# B&R Automation Studio project lab2
Automation Studio 4.5.2.102

## Configuration SampleText

CPU 4PP065.0571-P74, AutomationRuntime D4.52, Build 4.1.2, Vc V4.25.0, Safety 1.6

### Task classes (Cpu.sw)
```
Cyclic#1 (cycle 2000 us, tolerance 0 us):
  ncsdcctrl <- ncsdcctrl.prg
Cyclic#4:
  DoorCtrl <- DoorCtrl.prg
  LED <- LED.prg
DataObjects: Acp10sys
NcDataObjects: acp10etxen <- acp10etxen.dob, gAxis01a <- gAxis01obj.gAxis01a.dob, gAxis01i <- gAxis01obj.gAxis01i.dob
Binaries: TCData, udbdef, iomap, arconfig, asfw, ashwac, sysconf, User, Role, ashwd, acp10cfg, Acp10map
Libraries: Acp10sdc, sys_lib, Runtime, asstring, Acp10man, Acp10par, NcGlobal, Acp10_MC, brsystem, AsBrStr, GateCtrl, astime, fileio, powerlnk, asieccon
```

### Hardware
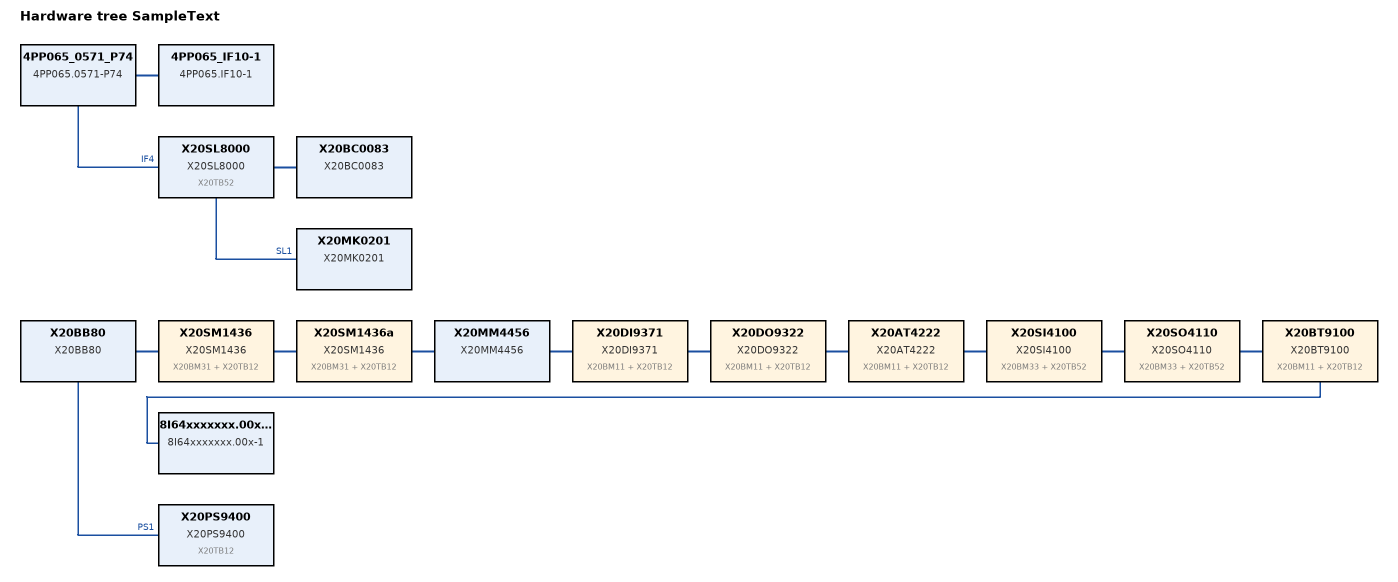
```
4PP065_0571_P74 : 4PP065.0571-P74 v1.1.2.0
  Connector IF4:
    EplInterfaceRedundant = 0
    EplEthInterfaceRedundant = 0
  Connector IF5:
    ActivateDevice = 1
    Mode = Manual
    InternetAddress = 10.0.1.1
    SubnetMask = 255.255.255.0
  ConfigurationID = labBR
  TimerDeviceType = EPLX2X
  TimerDevice = 4PP065_0571_P74.IF4
  TaskClassIdleTime = 2000
  Cyclic1Duration = 2000
  Cyclic1Tolerance = 0
  Cyclic1Output = 1
4PP065_IF10-1 : 4PP065.IF10-1 v1.0.3.0  [SS -> 4PP065_0571_P74.SS1]
8I64xxxxxxx.00x-1 : 8I64xxxxxxx.00x-1 v1.3.9.1  [X2X1 -> X20BT9100.X2X1 [Cable Type=X2XCable, Length=10, Version=1.0.0.2]]
  packedETAD = packed
  packedETI = packed
  packedCMDD = packed
  packedCMI = packed
  UNS = 220
  NCR = 10
  NSP = 890
  COS = 64
  RSC = 33000
X20AT4222 : X20AT4222 v1.2.3.0  [SS1 -> X20TB12e.SS; SL -> X20BM11c.SL1]
X20BB80 : X20BB80 v1.0.2.0
X20BC0083 : X20BC0083 v2.9.0.0  [PLK1 -> X20SL8000.PLK2 (NodeNumber=2) [Cable Type=PowerlinkCable, Length=10, Version=1.0.0.2]; SL -> X20BB80.SL1]
X20BM11 : X20BM11 v1.0.0.1  [X2X1 -> X20BM33a.X2X2]
X20BM11a : X20BM11 v1.0.0.1  [X2X1 -> X20MM4456.X2X2]
X20BM11b : X20BM11 v1.0.0.1  [X2X1 -> X20BM11a.X2X2]
X20BM11c : X20BM11 v1.0.0.1  [X2X1 -> X20BM11b.X2X2]
X20BM31 : X20BM31 v1.0.0.1  [X2X1 -> X20BB80.IF1]
X20BM31a : X20BM31 v1.0.0.1  [X2X1 -> X20BM31.X2X2]
X20BM33 : X20BM33 v1.0.0.4  [X2X1 -> X20BM11c.X2X2]
X20BM33a : X20BM33 v1.0.0.4  [X2X1 -> X20BM33.X2X2]
X20BT9100 : X20BT9100 v1.0.3.0  [SS1 -> X20TB12f.SS; SL -> X20BM11.SL1]
X20DI9371 : X20DI9371 v1.0.2.0  [SS1 -> X20TB12c.SS; SL -> X20BM11a.SL1]
X20DO9322 : X20DO9322 v1.0.3.0  [SS1 -> X20TB12d.SS; SL -> X20BM11b.SL1]
X20MK0201 : X20MK0201 v1.0.0.0  [SL -> X20SL8000.SL1]
X20MM4456 : X20MM4456 v1.1.5.0  [X2X1 -> X20BM31a.X2X2]
X20PS9400 : X20PS9400 v1.0.2.4  [SS1 -> X20TB12.SS; PS -> X20BB80.PS1]
X20SI4100 : X20SI4100 v1.10.1.1  [SS1 -> X20TB52.SS; SL -> X20BM33.SL1]
X20SL8000 : X20SL8000 v1.6.5.1  [PLK1 -> 4PP065_0571_P74.IF4 (NodeNumber=1) [Cable Type=PowerlinkCable, Length=10, Version=1.0.0.2]; PLK2 -> X20BC0083.PLK1 (NodeNumber=1) [Cable Type=PowerlinkCable, Length=10, Version=1.0.0.2]; SS1 -> X20TB52b.SS]
  SafeProject = SafeLOGIC-1
X20SM1436 : X20SM1436 v1.4.2.1  [SS1 -> X20TB12a.SS; SL -> X20BM31.SL1]
X20SM1436a : X20SM1436 v1.4.2.1  [SS1 -> X20TB12b.SS; SL -> X20BM31a.SL1]
X20SO4110 : X20SO4110 v1.10.1.1  [SS1 -> X20TB52a.SS; SL -> X20BM33a.SL1]
  SafeModuleID = 3
X20TB12 : X20TB12 v1.0.0.0
X20TB12a : X20TB12 v1.0.0.0
X20TB12b : X20TB12 v1.0.0.0
X20TB12c : X20TB12 v1.0.0.0
X20TB12d : X20TB12 v1.0.0.0
X20TB12e : X20TB12 v1.0.0.0
X20TB12f : X20TB12 v1.0.0.0
X20TB52 : X20TB52 v1.0.0.1
X20TB52a : X20TB52 v1.0.0.1
X20TB52b : X20TB52 v1.0.0.1
```

### IoMap.iom - 4PP065_0571_P74/IoMap.iom
```iecst
VAR_CONFIG
	Cyclic#1.gAxis01_DrvIf.iLifeCnt AT %IB."8I64xxxxxxx.00x-1".SDC_LifeCnt;
	Cyclic#1.gAxis01_DrvIf.iDrvOK AT %IX."8I64xxxxxxx.00x-1".ETAD_Input_Bool_02;
	Cyclic#1.gAxis01_DrvIf.oSetTime AT %QW."8I64xxxxxxx.00x-1".SDC_SetTime;
	Cyclic#1.::DoorCtrl:driveSM.speed AT %QW."8I64xxxxxxx.00x-1".LFRD_Output;
	Cyclic#1.gAxis01_DiDoIf.iLifeCntDriveReady AT %IB."8I64xxxxxxx.00x-1".SDC_LifeCnt;
	Cyclic#1.gAxis01_DiDoIf.iLifeCntDriveEnable AT %IB."8I64xxxxxxx.00x-1".SDC_LifeCnt;
	Cyclic#1.gAxis01_DiDoIf.oDriveEnable AT %QX."8I64xxxxxxx.00x-1".CMDD_Output_Bool_00;
	Cyclic#1.gAxis01_ModuleOk AT %QX."8I64xxxxxxx.00x-1".CMDD_Output_Bool_01;
	Cyclic#1.gAxis01_ModuleOk AT %QX."8I64xxxxxxx.00x-1".CMDD_Output_Bool_02;
	Cyclic#1.gAxis01_ModuleOk AT %IX."8I64xxxxxxx.00x-1".ModuleOk;
	Cyclic#1.gAxis01_DiDoIf.oDriveEnable AT %QX."8I64xxxxxxx.00x-1".CMDD_Output_Bool_03;
	Cyclic#1.gAxis01_DiDoIf.iDriveReady AT %IX."8I64xxxxxxx.00x-1".ETAD_Input_Bool_02;
	::DoorCtrl:doorSM.direction AT %IX."X20DI9371".DigitalInput01;
	::DoorCtrl:doorSM.sw1 AT %IX."X20DI9371".DigitalInput02;
	::DoorCtrl:doorSM.sw2 AT %IX."X20DI9371".DigitalInput03;
	::DoorCtrl:doorSM.sw3 AT %IX."X20DI9371".DigitalInput04;
	::DoorCtrl:doorSM.sw4 AT %IX."X20DI9371".DigitalInput05;
	::LED:Led1 AT %QX."X20DO9322".DigitalOutput02;
	::LED:Led2 AT %QX."X20DO9322".DigitalOutput03;
	::LED:Led3 AT %QX."X20DO9322".DigitalOutput04;
	::LED:Led4 AT %QX."X20DO9322".DigitalOutput05;
	::DoorCtrl:driveSM.state  AT %IW."8I64xxxxxxx.00x-1".ETAD_Input;
	::DoorCtrl:driveSM.command  AT %QW."8I64xxxxxxx.00x-1".CMDD_Output;
END_VAR
```

## Logical view

Binary libraries used (declarations not repeated): Runtime, Operator, AsIecCon, astime, sys_lib, asstring, Acp10man, Acp10par, NcGlobal, Acp10sdc, Acp10_MC, brsystem, AsBrStr

### Global.var - Global variables
```iecst
VAR
	gAxis01 : ACP10AXIS_typ := (0);
	gAxis01_HW : SdcHwCfg_typ := (0);
	gAxis01_DrvIf : SdcDrvIf16_typ := (0);
	gAxis01_DiDoIf : SdcDiDoIf_typ := (0);
	gAxis01_ModuleOk : BOOL := 0;
	L1 : BOOL;
	L2 : BOOL;
	L3 : BOOL;
	L4 : BOOL;
END_VAR
```

### Package Logical/Libraries - Global libraries

### Library Logical/Libraries/GateCtrl (ANSIC)

#### Types.typ - Exported data types
```iecst
TYPE
	GateState :
		(
		ST_INIT := 0,
		ST_UNKNOWN := 1,
		ST_OPEN := 2,
		ST_CLOSE := 3,
		ST_ACC_POS := 4,
		ST_ACC_NEG := 5,
		ST_POS := 6,
		ST_NEG := 7,
		ST_DEC_POS := 8,
		ST_DEC_NEG := 9
		);
	drivecommand :
		(
		CMD_SWITCHED_ON := 7,
		CMD_ENABLE := 15,
		CMD_SHUTDOWN := 6,
		STATE_READY := 33,
		STATE_DISABLED := 64,
		STATE_SWITCHED_ON := 35
		);
END_TYPE
```

#### GateCtrl.fun - Exported functions and function blocks
```iecst
{REDUND_ERROR} {REDUND_UNREPLICABLE} FUNCTION_BLOCK DoorStateMachine (*TODO: Add your comment here*) (*$GROUP=User,$CAT=User,$GROUPICON=User.png,$CATICON=User.png*)
	VAR_INPUT
		state : {REDUND_UNREPLICABLE} GateState;
		sw1 : {REDUND_UNREPLICABLE} BOOL;
		sw2 : {REDUND_UNREPLICABLE} BOOL;
		sw3 : {REDUND_UNREPLICABLE} BOOL;
		sw4 : {REDUND_UNREPLICABLE} BOOL;
		direction : {REDUND_UNREPLICABLE} BOOL;
	END_VAR
	VAR_OUTPUT
		speed : {REDUND_UNREPLICABLE} INT;
	END_VAR
	VAR
		swo1 : {REDUND_UNREPLICABLE} USINT;
		swo2 : {REDUND_UNREPLICABLE} USINT;
		swo3 : {REDUND_UNREPLICABLE} USINT;
		swo4 : {REDUND_UNREPLICABLE} USINT;
	END_VAR
END_FUNCTION_BLOCK

{REDUND_ERROR} FUNCTION_BLOCK LedStateMachine (*TODO: Add your comment here*) (*$GROUP=User,$CAT=User,$GROUPICON=User.png,$CATICON=User.png*)
	VAR_INPUT
		state : {REDUND_UNREPLICABLE} GateState;
	END_VAR
	VAR_OUTPUT
		led1 : {REDUND_UNREPLICABLE} BOOL;
		led2 : {REDUND_UNREPLICABLE} BOOL;
		led3 : {REDUND_UNREPLICABLE} BOOL;
		led4 : {REDUND_UNREPLICABLE} BOOL;
		timer : INT;
	END_VAR
END_FUNCTION_BLOCK

{REDUND_ERROR} {REDUND_UNREPLICABLE} FUNCTION_BLOCK DriveStateMachine (*TODO: Add your comment here*) (*$GROUP=User,$CAT=User,$GROUPICON=User.png,$CATICON=User.png*)
	VAR_INPUT
		enable : {REDUND_UNREPLICABLE} BOOL;
		state : {REDUND_UNREPLICABLE} UINT;
	END_VAR
	VAR_OUTPUT
		speed : {REDUND_UNREPLICABLE} INT;
		command : {REDUND_UNREPLICABLE} UINT;
	END_VAR
END_FUNCTION_BLOCK
```

#### DoorStateMachine.c
```c
#include <bur/plctypes.h>
#ifdef __cplusplus
	extern "C"
	{
#endif
	#include "GateCtrl.h"
#ifdef __cplusplus
	};
#endif
/* TODO: Add your comment here */
void DoorStateMachine(struct DoorStateMachine* inst)
{
	/*TODO: Add your code here*/
	switch(inst->state)
	{
		case ST_INIT:
			{
				if(inst->sw1==0 && inst->sw2==0 && inst->sw3==0 && inst->sw4==0)
					inst->state=ST_UNKNOWN;
				break;
			}
		case ST_UNKNOWN:
			{
				if(inst->direction==1 && inst->sw1!=inst->swo1)
					inst->state=ST_CLOSE;
				if(inst->direction==0 && inst->sw4!=inst->swo4)
					inst->state=ST_OPEN;
				break;
			}
		case ST_CLOSE:
			{
				inst->speed = 0;
				if(inst->direction==1 && inst->sw1!=inst->swo1)
					inst->state=ST_ACC_NEG;
				break;//
			}
		case ST_ACC_NEG:
			{
				inst->speed = -200;
				if(inst->direction==1 && inst->sw2!=inst->swo2)
					inst->state=ST_NEG;
				if(inst->direction==0)
					inst->state=ST_DEC_POS;
				break;

			}
		case ST_NEG:
			{
				inst->speed = -600;
				if(inst->direction==1 && inst->sw3!=inst->swo3)
					inst->state=ST_DEC_NEG;
				if(inst->direction==0)
					inst->state=ST_POS;
				break;
			}
		case ST_DEC_NEG:
			{

				inst->speed = -200;
				if(inst->direction==1 && inst->sw4!=inst->swo4)
					inst->state=ST_OPEN;
				break;
			}

		case ST_OPEN:
			{
				inst->speed = 0;
				if(inst->direction==0 && inst->sw4!=inst->swo4)
					inst->state=ST_ACC_POS;
				break;
			}
		case ST_ACC_POS:
			{
				inst->speed = 200;
				if(inst->direction==0 && inst->sw3!=inst->swo3)
					inst->state=ST_POS;
				if(inst->direction==1)
					inst->state=ST_DEC_NEG;
				break;
			}
		case ST_POS:
			{
				inst->speed = 600;
				if(inst->direction==0 && inst->sw2!=inst->swo2)
					inst->state=ST_DEC_POS;
				if(inst->direction==1)
					inst->state=ST_NEG;
				break;
			}
		case ST_DEC_POS:
			{
				inst->speed = 200;
				if(inst->direction==0 && inst->sw1!=inst->swo1)
					inst->state=ST_CLOSE;
				break;
			}
	}
	inst->swo1 = inst->sw1;
	inst->swo2 = inst->sw2;
	inst->swo3 = inst->sw3;
	inst->swo4 = inst->sw4;
}
```

#### LedStateMachine.c
```c
#include <bur/plctypes.h>
#ifdef __cplusplus
	extern "C"
	{
#endif
#include "GateCtrl.h"
#ifdef __cplusplus
	};
#endif
/* TODO: Add your comment here */
void LedStateMachine(struct LedStateMachine* inst)
{
	{
		/*TODO: Add your code here*/
		switch(inst->state)
		{
			case ST_INIT:
				{
					inst->led1 = 0 ;
					inst->led2 = 0 ;
					inst->led3 = 0 ;
					inst->led4 = 0 ;
					break;
				}
			case ST_UNKNOWN:
				{
					if(inst->timer%10==0)
					{
						inst->led1 = !inst->led1;
						inst->led2 = !inst->led2;
						inst->led3 = !inst->led3;
						inst->led4 = !inst->led4;
					}
					break;
				}
			case ST_CLOSE:
				{

					inst->led1 = 1;
					inst->led2 = 1;
					inst->led3 = 1;
					inst->led4 = 1;
					break;
				}

			case ST_ACC_NEG:
				{

					inst->led1 = 0;
					inst->led2 = 1;
					inst->led3 = 1;
					inst->led4 = 1;
					break;
				}
			case ST_NEG:
				{

					inst->led1 = 0;
					inst->led2 = 0;
					inst->led3 = 1;
					inst->led4 = 1;
					break;
				}
			case ST_DEC_NEG:
				{

					inst->led1 = 0;
					inst->led2 = 0;
					inst->led3 = 0;
					inst->led4 = 1;
					break;
				}

			case ST_OPEN:
				{

					inst->led1 = 0;
					inst->led2 = 0;
					inst->led3 = 0;
					inst->led4 = 0;
					break;
				}

			case ST_ACC_POS:
				{

					inst->led1 = 0;
					inst->led2 = 0;
					inst->led3 = 0;
					inst->led4 = 1;
					break;
				}
			case ST_POS:
				{

					inst->led1 = 0;
					inst->led2 = 0;
					inst->led3 = 1;
					inst->led4 = 1;
					break;
				}
			case ST_DEC_POS:
				{

					inst->led1 = 0;
					inst->led2 = 1;
					inst->led3 = 1;
					inst->led4 = 1;
					break;
				}
		}
	}
	//inst->timer++;
}
```

#### DriveStateMachine.c
```c
#include <bur/plctypes.h>
#ifdef __cplusplus
extern "C"
{
#endif
#include "GateCtrl.h"
#ifdef __cplusplus
};
#endif
void DriveStateMachine (struct DriveStateMachine* inst)
{
	UINT mask = inst->state & 0x6f;
	if(!inst->enable)
	{
		inst->command = CMD_SHUTDOWN;
	}
	else
	{
		switch (mask)
		{
			//Выключенный двигатель
			case STATE_DISABLED:
				inst->command = CMD_SHUTDOWN;
				break;
			//Включенный двигатель
			case STATE_SWITCHED_ON:
				inst->command = CMD_SWITCHED_ON;
				break;
			//Готовый двигатель
			case STATE_READY:
				inst->command = CMD_ENABLE;
				break;
		}
	}
}
```

### Program Logical/DoorCtrl (ANSIC)

#### Variables.var
```iecst
VAR
	doorSM : DoorStateMachine := (0);
	ledSM : LedStateMachine := (0);
	ETAD : UINT := 0;
	Speed : INT := 0;
	driveSM : DriveStateMachine;
END_VAR
```

#### Main.cpp
```cpp
#include <bur/plctypes.h>

#ifdef _DEFAULT_INCLUDES
	#include <AsDefault.h>
#endif

// amount of memory to be allocated for heap storage must be specified for every ANSI C++ program with the bur_heap_size variable
unsigned long bur_heap_size = 0xFFFF;

void _INIT ProgramInit(void)
{
	driveSM.enable = 1;	// Insert code here

}

void _CYCLIC ProgramCyclic(void)
{
	DoorStateMachine (&doorSM);
	driveSM.speed=doorSM.speed;
	DriveStateMachine(&driveSM);
	ledSM.state = doorSM.state;
	LedStateMachine(&ledSM);
	L1=ledSM.led1;
	L2=ledSM.led2;
	L3=ledSM.led3;
	L4=ledSM.led4;
}

void _EXIT ProgramExit(void)
{
	// Insert code here

}
```

### Program Logical/LED (ANSIC)

#### Variables.var
```iecst
VAR
	Led : LedStateMachine;
	Led1 : BOOL;
	Led2 : BOOL;
	Led3 : BOOL;
	Led4 : BOOL;
END_VAR
```

#### Main.cpp
```cpp
#include <bur/plctypes.h>

#ifdef _DEFAULT_INCLUDES
	#include <AsDefault.h>
#endif

// amount of memory to be allocated for heap storage must be specified for every ANSI C++ program with the bur_heap_size variable
unsigned long bur_heap_size = 0xFFFF;

void _INIT ProgramInit(void)
{
	// Insert code here

}

void _CYCLIC ProgramCyclic(void)
{
	LedStateMachine(&Led);

		Led1 = L1;
		Led2 = L2;
		Led3 = L3;
		Led4 = L4;
}

void _EXIT ProgramExit(void)
{
	// Insert code here

}
```

Listed in the project but not available here: Logical/Global.typ, Logical/Libraries/GateCtrl/Constants.var, Logical/ncsdcctrl, Logical/acp10etxen, Logical/gAxis01obj
